FUNCTION_BLOCK FB_DeviceReal EXTENDS FB_LinkDataReal
VAR_INPUT		
	nControl  			: BYTE;
	fControlData  		: REAL;
END_VAR

VAR_OUTPUT
	nStatus  			: BYTE;
	fStatusData  		: REAL;
END_VAR

SUPER^();
Control := nControl;
ControlData := fControlData;
nStatus := Status;
fStatusData := StatusData;

END_FUNCTION_BLOCK

(* stored: Version 1.1.0.1, ProductVersion 3.1.4024.12
   POU FB_DeviceReal: Id {87a52e17-6f15-0348-1881-2797e6232087}, SpecialFunc None *)
